Staubli VAL3: motionStatus.pgx

public program motionStatus(num x_nInConnFlag)
begin

  // Do nothing
  // See start() program for more details

end
